Yaskawa INFORM job: R1_W27-A2(90,-90)POPR-KM-OK_MOD.JBI

/JOB
//NAME R1_W27-A2(90,-90)POPR-KM-OK_MOD
///FOLDERNAME KRIS-SCIANA
//POS
///NPOS 183,183,0,6,0,0
///TOOL 0
///POSTYPE PULSE
///PULSE
C00000=47255,92390,21974,-39561,97708,85383
C00001=10855,-90008,-88389,-33686,75537,85808
C00002=-111602,-139258,-125525,-5527,77988,-30584
C00003=-111602,-139258,-125525,-5527,77988,-30584
C00004=-63451,-99780,-87259,-34493,107645,-18593
C00005=-79235,-87779,-71168,-36428,98005,-22127
C00006=-81155,-88041,-68185,-36487,95587,-22123
C00007=-83679,-90006,-68978,-36755,94086,-22676
C00008=-83320,-89737,-68871,-36718,94298,-22597
C00009=-83320,-90271,-70181,-36754,94730,-22742
C00010=-84421,-91093,-70507,-36864,94080,-22984
C00011=-84421,-90731,-69628,-36842,93792,-22887
C00012=-81728,-89912,-71997,-36675,96467,-22659
C00013=-111602,-139258,-125525,-5527,77988,-30584
C00014=-111602,-139258,-125525,-5527,77988,-30584
C00015=-131748,-141016,-124490,10531,76516,-37016
C00016=-120565,-128207,-90021,8850,60749,-34228
C00017=-114295,-127384,-89205,7232,60054,-31882
C00018=-112834,-127008,-88848,6844,59902,-31333
C00019=-110412,-126666,-88756,6184,59829,-30410
C00020=-111525,-126835,-88802,6488,59856,-30835
C00021=-111525,-128465,-91197,6450,60489,-30798
C00022=-108910,-128023,-91079,5736,60447,-29805
C00023=-108910,-126871,-89375,5761,59994,-29827
C00024=-114109,-129808,-92766,7120,60979,-31753
C00025=-125724,-137992,-104372,9805,65099,-35816
C00026=-168598,-158328,-94882,65934,65859,5142
C00027=-138330,-90233,-84655,36621,76479,52498
C00028=-128715,-49536,-61129,33505,77884,56923
C00029=-128662,-48132,-55305,33830,75458,56202
C00030=-128776,-48721,-53911,34016,74532,55864
C00031=-127610,-48935,-54036,33707,74044,56192
C00032=-128384,-48797,-53955,33914,74367,55973
C00033=-127721,-49153,-57529,33460,75800,56690
C00034=-129344,-26255,-35376,41772,85568,55954
C00035=-129502,-28873,-35296,41846,84590,55492
C00036=-129628,-31082,-36795,41874,84489,55393
C00037=-129540,-29583,-35781,41856,84558,55460
C00038=-128070,-29028,-37630,41593,84938,56269
C00039=-125732,-38818,-42817,41353,82441,56314
C00040=-125732,-38715,-41972,41387,82085,56171
C00041=-125732,-38825,-42888,41351,82471,56325
C00042=-132576,-10372,-23557,42183,87769,55412
C00043=-126022,-12465,-28572,31920,86751,56828
C00044=-125240,-12576,-28656,31787,86457,57050
C00045=-126011,-12468,-28573,31917,86746,56832
C00046=-125354,-12526,-30294,30962,87436,57184
C00047=-120977,-16940,-33250,30218,85489,58339
C00048=-121063,-17240,-32162,30257,84802,58123
C00049=-121058,-15104,-30561,30253,84897,58149
C00050=-121061,-16554,-31651,30256,84834,58131
C00051=-121060,-15778,-32671,30227,85727,58368
C00052=-117907,-13652,-30768,29609,84558,59259
C00053=-117907,-13692,-29869,29630,84054,59130
C00054=-117057,-13593,-30324,29443,84053,59453
C00055=-124504,-18943,-37628,40859,87235,58732
C00056=-122503,-58034,-63350,23085,92729,-39111
C00057=-118561,-36204,-48728,23381,102965,-35613
C00058=-118381,-37612,-47396,23227,101492,-35840
C00059=-119514,-54944,-57534,22827,90064,-38535
C00060=-118197,-55011,-58807,22737,90395,-37994
C00061=-117359,-61105,-60828,21568,85220,-34341
C00062=-119392,-54872,-58672,22830,90711,-38368
C00063=-122456,-57021,-66004,23167,94704,-38710
C00064=-79548,-70371,-81102,-16241,84903,14397
C00065=-79548,-70265,-68951,-16505,77767,15353
C00066=-104563,-100291,-63220,13387,32000,-19094
C00067=-104975,-100452,-63184,13820,31966,-19359
C00068=-115302,-93136,-62932,26704,43721,-31733
C00069=-113448,-91077,-63180,22011,45608,-32160
C00070=-114452,-94731,-67163,22359,46409,-32454
C00071=-99886,-76150,-67523,500,65373,-23503
C00072=-75740,-68220,-64202,-17439,76767,16862
C00073=-76507,-66361,-64522,-17207,77706,16451
C00074=-95900,-77133,-67906,-2885,65671,-13753
C00075=-83981,-71880,-65491,-14621,70935,-768
C00076=-83123,-70857,-64909,-14849,71253,-493
C00077=-81635,-70718,-66741,-15162,72688,-135
C00078=-81323,-43477,-57369,-10673,89641,51992
C00079=-82758,-42773,-53931,-10445,87732,51670
C00080=-82626,-42173,-53561,-10465,87828,51707
C00081=-82621,-41471,-53126,-10465,87921,51700
C00082=-92310,-5151,-28231,-6661,90278,58032
C00083=-92716,-2727,-26257,-6592,90277,57898
C00084=-95848,18216,-9468,-2153,101928,56962
C00085=-96696,22336,-5572,-2620,102588,67876
C00086=-92622,2167,-26871,-6629,93158,57779
C00087=-102765,8643,-22555,7262,102808,72751
C00088=-102913,11884,-15167,7450,102139,72741
C00089=-104434,11036,-15928,7485,102306,72236
C00090=-104019,13462,-16416,6672,103835,72468
C00091=-100362,7840,-23814,352,99133,73837
C00092=-93505,-42567,-98732,-7157,86742,74535
C00093=-125724,-137992,-104372,9805,65099,-35816
C00094=-110950,-137574,-92834,6542,56798,-30799
C00095=-108633,-136098,-91409,5901,56506,-29909
C00096=-110317,-120133,-87198,6027,62209,-30244
C00097=-115536,-122151,-89589,7364,63072,-32157
C00098=-115536,-142518,-126484,6818,75223,-31432
C00099=-115536,-142518,-126484,6818,75223,-31432
C00100=27632,69086,-255,32308,94480,64498
C00101=22775,131727,30764,-8837,96794,84364
C00102=23208,121491,44257,-39062,86083,83812
C00103=-45129,13731,-11238,-25738,101470,44798
C00104=-54749,18539,-6974,-25294,98453,41899
C00105=-54749,18238,-2799,-25102,95977,42433
C00106=-54749,18226,-2184,-25080,95627,42508
C00107=-54749,18240,-2936,-25107,96054,42417
C00108=-50930,35725,13913,-25203,95936,43853
C00109=-64523,30372,3224,-1874,95567,42430
C00110=-64687,29964,2819,-1861,95602,42375
C00111=-65096,28955,1821,-1825,95689,42236
C00112=-64964,29394,1262,-1838,96260,42271
C00113=-65321,28613,-146,-1811,96720,42147
C00114=-68202,27629,-336,-1561,96271,41197
C00115=-68113,27223,145,-1567,95770,41232
C00116=-67724,25933,-1111,-1601,95888,41360
C00117=-68202,27629,-336,-1561,96271,41197
C00118=-69952,33819,5307,-1407,95949,40620
C00119=-71494,37291,10752,-1268,94359,40124
C00120=-71910,38959,12475,-1230,94150,39986
C00121=-71687,38230,9822,-1254,95411,40047
C00122=-69715,46382,18396,-1423,94355,40716
C00123=-70085,45287,18762,-1387,93560,40601
C00124=-70403,44519,17944,-1360,93663,40494
C00125=-69715,46382,18396,-1423,94355,40716
C00126=-70506,44470,16366,-1355,94608,40450
C00127=-74342,36127,7664,-1021,95621,39166
C00128=-67594,51845,26562,-12944,100620,40046
C00129=-67594,51857,27602,-12911,100003,40111
C00130=-67594,51846,26389,-12950,100725,40035
C00131=-74342,37093,2887,-1031,99056,39137
C00132=-67920,8103,-14728,-23481,111043,54078
C00133=-68371,9278,-10792,-23231,109243,54283
C00134=-71989,6025,-15002,-18365,107550,55075
C00135=-68543,9839,-10380,-23257,109228,54219
C00136=-67871,11157,-7953,-23050,108659,54597
C00137=-70618,6902,-11763,-25009,100838,46496
C00138=-68309,7669,-17399,-25439,105035,46441
C00139=-35319,67510,50034,-36864,102833,41158
C00140=-36426,60496,49514,-37352,95882,39315
C00141=-36245,61460,50947,-37306,95650,39472
C00142=-37635,75219,67177,-34434,97406,42519
C00143=-35605,73747,62011,-36095,100000,42690
C00144=-48748,75637,44138,-12559,109446,36491
C00145=-47018,7632,-18403,-16315,86685,22647
C00146=-48186,9094,-11222,-16117,82930,22742
C00147=-48900,12300,-7759,-15972,82326,22576
C00148=-48845,10311,-10218,-15969,82810,22529
C00149=-48144,8977,-10156,-16147,82248,22846
C00150=-48792,12294,-7764,-15997,82346,22611
C00151=-48554,12497,-7580,-16051,82384,22689
C00152=-47807,15110,-5208,-16221,82416,22944
C00153=-47830,15796,-4582,-16217,82378,22941
C00154=-47157,14640,-7349,-16336,83577,23014
C00155=-46490,6362,-16531,-16455,85053,23045
C00156=-51089,14800,-9249,10241,81305,-15900
C00157=-51639,15771,-6503,10417,80201,-16178
C00158=-51452,17933,-2732,10403,78988,-16218
C00159=-52394,14452,-5453,10658,78994,-16538
C00160=-51853,16186,-5099,10493,79587,-16303
C00161=-61783,45784,25403,13194,77537,-19938
C00162=-67433,89838,76993,23343,85040,-43070
C00163=-67406,90447,77765,23345,84883,-43090
C00164=-67651,91444,77676,23339,85475,-43066
C00165=-51787,16236,-7953,10429,81332,-16133
C00166=-102783,1332,-28831,-2508,120082,-77442
C00167=-102957,2789,-26573,-2528,119437,-77492
C00168=-103006,2286,-25832,-2518,118722,-77496
C00169=-103017,3676,-26663,-2555,119947,-77527
C00170=-103226,5472,-23865,-2576,119142,-77587
C00171=-101649,3064,-25171,-2232,118754,-76984
C00172=-101836,5087,-24653,-2291,119469,-77071
C00173=-102782,1324,-28838,-2508,120083,-77442
C00174=-102716,1959,-28722,-3690,98810,-77621
C00175=-111602,-139258,-125525,-5527,77988,-30584
C00176=-63451,-99780,-87259,-34493,107645,-18593
C00177=-77664,-93447,-72354,-35997,96893,-21092
C00178=-71109,-84007,-59579,-44165,102740,-19972
C00179=-76711,-72421,-54458,-45861,101920,-22309
C00180=-73740,-70290,-55538,-45661,104697,-22163
C00181=-73778,-73289,-89979,-52376,117942,-29543
C00182=4604,-97136,-110463,-3690,98810,-77621
BC00000=173361,170327,1069948
BC00001=285044,126360,1057855
BC00002=197925,2384,1013850
BC00003=398093,2384,1013850
BC00004=398093,2384,1013850
BC00005=398093,2384,1013850
BC00006=398093,2384,1013850
BC00007=398093,2384,1013850
BC00008=398093,2384,1013850
BC00009=398093,2384,1013850
BC00010=398093,2384,1013850
BC00011=398093,2384,1013850
BC00012=398093,2384,1013850
BC00013=398093,2384,1013850
BC00014=197925,2384,1013850
BC00015=16093,2384,1007970
BC00016=16093,2384,1007970
BC00017=16093,2384,1007970
BC00018=16093,2384,1007970
BC00019=16093,2384,1007970
BC00020=16093,2384,1007970
BC00021=16093,2384,1007970
BC00022=16093,2384,1007970
BC00023=16093,2384,1007970
BC00024=16093,2384,1007970
BC00025=16093,2384,1007970
BC00026=2663,3711,1022453
BC00027=269,7512,1047096
BC00028=269,7512,1047096
BC00029=269,7512,1047096
BC00030=269,7512,1047096
BC00031=269,7512,1047096
BC00032=269,7512,1047096
BC00033=269,7512,1047096
BC00034=15,11820,1075020
BC00035=15,11820,1075020
BC00036=15,11820,1075020
BC00037=15,11820,1075020
BC00038=15,11820,1075020
BC00039=15,11820,1075020
BC00040=15,11820,1075020
BC00041=15,11820,1075020
BC00042=15,11820,1075020
BC00043=15,11820,1075020
BC00044=15,11820,1075020
BC00045=15,11820,1075020
BC00046=15,11820,1075020
BC00047=15,11820,1075020
BC00048=15,11820,1075020
BC00049=15,11820,1075020
BC00050=15,11820,1075020
BC00051=15,11820,1075020
BC00052=15,11820,1075020
BC00053=15,11820,1075020
BC00054=15,11820,1075020
BC00055=15,11820,1075020
BC00056=15,49099,1075175
BC00057=15,47349,1075175
BC00058=15,47349,1075175
BC00059=15,47349,1075175
BC00060=15,47349,1075175
BC00061=15,62077,1075175
BC00062=15,62577,1075175
BC00063=15,63827,1075175
BC00064=15,12213,1075175
BC00065=15,12213,1075175
BC00066=16,12213,1075171
BC00067=16,12213,1075171
BC00068=16,12213,1075171
BC00069=16,12213,1075171
BC00070=16,12213,1075171
BC00071=16,12213,1075171
BC00072=15,16755,1075175
BC00073=15,16755,1075175
BC00074=16,12213,1075171
BC00075=16,12213,1075171
BC00076=16,12213,1075171
BC00077=16,12213,1075171
BC00078=16,12213,1075171
BC00079=16,12213,1075171
BC00080=16,12213,1075171
BC00081=16,12213,1075171
BC00082=16,12213,1075171
BC00083=16,12213,1075171
BC00084=16,12213,1075171
BC00085=16,12213,1075171
BC00086=16,12213,1075171
BC00087=17,22433,1075169
BC00088=17,22433,1075167
BC00089=17,22433,1075167
BC00090=17,22433,1075169
BC00091=16,12213,1075171
BC00092=16,12213,1075171
BC00093=16093,2384,1007970
BC00094=16093,2384,1007970
BC00095=16093,2384,1007970
BC00096=16093,2384,1007970
BC00097=16093,2384,1007970
BC00098=16093,2384,1007970
BC00099=92875,102,1007970
BC00100=25030,15919,1060143
BC00101=103306,16446,1075157
BC00102=79646,13110,1075161
BC00103=246913,5043,1075175
BC00104=246913,5043,1075175
BC00105=246913,5043,1075175
BC00106=246913,5043,1075175
BC00107=246913,5043,1075175
BC00108=246913,5043,1075175
BC00109=246913,5043,1075175
BC00110=246913,5043,1075175
BC00111=246913,5043,1075175
BC00112=246913,5043,1075175
BC00113=246913,5043,1075175
BC00114=246913,5043,1075175
BC00115=246913,5043,1075175
BC00116=246913,5043,1075175
BC00117=246913,5043,1075175
BC00118=246913,5043,1075175
BC00119=246913,5043,1075175
BC00120=246913,5043,1075175
BC00121=246913,5043,1075175
BC00122=246913,5043,1075175
BC00123=246913,5043,1075175
BC00124=246913,5043,1075175
BC00125=246913,5043,1075175
BC00126=246913,5043,1075175
BC00127=246913,5043,1075175
BC00128=246913,5043,1075175
BC00129=246913,5043,1075175
BC00130=246913,5043,1075175
BC00131=246913,5043,1075175
BC00132=310215,25331,1075175
BC00133=304559,24148,1075175
BC00134=304559,24148,1075175
BC00135=302296,23674,1075175
BC00136=302296,23674,1075175
BC00137=304559,24148,1075175
BC00138=304559,24148,1075175
BC00139=197323,15,1075175
BC00140=197323,15,1075175
BC00141=197323,15,1075175
BC00142=197323,15,1075175
BC00143=197323,15,1075175
BC00144=197323,15,1075175
BC00145=197986,15,1075175
BC00146=197986,15,1075175
BC00147=198112,15,1075175
BC00148=198252,15,1075175
BC00149=198252,15,1075175
BC00150=198112,15,1075175
BC00151=198112,15,1075175
BC00152=198112,15,1075175
BC00153=198112,15,1075175
BC00154=198112,15,1075175
BC00155=199434,15,1075175
BC00156=148787,33401,1075175
BC00157=154351,32151,1075175
BC00158=155733,31841,1075173
BC00159=156576,31651,1075175
BC00160=156576,31651,1075175
BC00161=155733,31841,1075173
BC00162=155733,31841,1075173
BC00163=155733,31841,1075173
BC00164=155733,31841,1075173
BC00165=148927,71500,1075175
BC00166=344706,64580,1052547
BC00167=343940,58320,1037184
BC00168=343871,57754,1035794
BC00169=343634,55816,1031039
BC00170=343634,55816,1031039
BC00171=343871,57754,1035794
BC00172=343871,57754,1035794
BC00173=341638,64598,1052619
BC00174=341637,64597,1052617
BC00175=398093,160168,1013850
BC00176=398093,2384,1013850
BC00177=398093,2384,1013850
BC00178=398093,2384,1013850
BC00179=398093,2384,1013850
BC00180=398093,2384,1013850
BC00181=398093,2384,1013850
BC00182=176985,505314,1052617
///POSTYPE BASE
///RECTAN
///RCONF 0,0,0,0,1,0,0,0,0,0,0,0,0,0,0,0,0,0,0,0,0,0,0,0
P00006=2.006,1.622,-0.565,0.0000,0.0000,0.0000
///RCONF 0,0,0,0,0,0,0,0,0,0,0,0,0,0,0,0,0,0,0,0,0,0,0,0
P00023=-2.957,-4.083,2.762,0.0000,0.0000,0.0000
P00024=-1.466,-0.226,-0.419,0.0000,0.0000,0.0000
P00025=3.643,0.007,-2.585,0.0000,0.0000,0.0000
P00040=2.716,-0.016,3.014,0.0000,0.0000,0.0000
P00041=-0.109,0.014,0.966,0.0000,0.0000,0.0000
//INST
///DATE 2025/01/17 12:20
///ATTR SC,RW
///GROUP1 RB1,BS1
NOP
SFTOF
MOVJ C00000 BC00000 VJ=100.00
MOVJ C00001 BC00001 VJ=100.00
MOVJ C00002 BC00002 VJ=100.00
'DODANO BP 060624
MOVJ C00003 BC00003 VJ=100.00
MOVJ C00004 BC00004 VJ=100.00
MOVL C00005 BC00005 V=233.3
MOVL C00006 BC00006 V=60.0
REFP 3 C00007 BC00007
CALL JOB:SEARCH-R1
SET P040 P006
SFTON P040
MOVL C00008 BC00008 V=100.0
MOVL C00009 BC00009 V=100.0
MOVL C00010 BC00010 V=60.0
REFP 3 C00011 BC00011
CALL JOB:SEARCH-R1
SET P040 P006
SFTON P040
MOVL C00012 BC00012 V=100.0
MOVJ C00013 BC00013 VJ=100.00
MOVJ C00014 BC00014 VJ=100.00
MOVL C00015 BC00015 V=666.7
MOVL C00016 BC00016 V=666.7
MOVL C00017 BC00017 V=233.3
MOVL C00018 BC00018 V=60.0
REFP 3 C00019 BC00019
CALL JOB:SEARCH-R1
SET P041 P006
SFTON P041
MOVL C00020 BC00020 V=100.0
MOVL C00021 BC00021 V=100.0
MOVL C00022 BC00022 V=60.0
REFP 3 C00023 BC00023
CALL JOB:SEARCH-R1
SET P041 P006
SFTON P041
MOVL C00024 BC00024 V=100.0
MOVL C00025 BC00025 V=666.7
'KONIEC BP 060624
MOVJ C00026 BC00026 VJ=100.00
MOVJ C00027 BC00027 VJ=100.00
MOVJ C00028 BC00028 VJ=100.00
MOVJ C00029 BC00029 VJ=100.00
MOVL C00030 BC00030 V=60.0
REFP 3 C00031 BC00031
CALL JOB:SEARCH-R1
SET P023 P006
SFTON P023
MOVL C00032 BC00032 V=60.0
MOVL C00033 BC00033 V=100.0
MOVL C00034 BC00034 V=100.0
MOVL C00035 BC00035 V=100.0
REFP 3 C00036 BC00036
CALL JOB:SEARCH-R1
SET P023 P006
SFTON P023
MOVL C00037 BC00037 V=60.0
MOVL C00038 BC00038 V=100.0
MOVL C00039 BC00039 V=100.0
REFP 3 C00040 BC00040
CALL JOB:SEARCH-R1
SET P023 P006
SFTON P023
MOVL C00041 BC00041 V=60.0
'DRUGI NOWY POMIAR
SFTOF
MOVL C00042 BC00042 V=100.0
MOVL C00043 BC00043 V=100.0
REFP 3 C00044 BC00044
CALL JOB:SEARCH-R1
SET P024 P006
SFTON P024
MOVL C00045 BC00045 V=60.0
MOVL C00046 BC00046 V=100.0
MOVL C00047 BC00047 V=100.0
MOVL C00048 BC00048 V=60.0
REFP 3 C00049 BC00049
CALL JOB:SEARCH-R1
SET P024 P006
SFTON P024
MOVL C00050 BC00050 V=60.0
MOVL C00051 BC00051 V=100.0
MOVL C00052 BC00052 V=60.0
REFP 3 C00053 BC00053
CALL JOB:SEARCH-R1
SET P024 P006
SFTON P024
MOVL C00054 BC00054 V=60.0
MOVJ C00055 BC00055 VJ=30.00
SFTOF
COMM 'Path W988
COMM SFTOF
COMM SFTON P023
COMM CALL JOB:COFNIJ_DRUT
COMM MOVJ C00056 BC00056 VJ=50.00
COMM MOVJ C00057 BC00057 VJ=100.00
COMM MOVL C00058 BC00058 V=100.0 PL=0
COMM REFP 1 C00059 BC00059
COMM REFP 2 C00060 BC00060
COMM MACRO1 MJ#(0) ARGF7
COMM ARCON
COMM SFTON P024
COMM MOVL C00061 BC00061 V=10.8
COMM ARCOF
COMM MOVL C00062 BC00062 V=100.0
COMM MOVJ C00063 BC00063 VJ=50.00
COMM SFTOF
COMM 'Path W989
COMM SFTOF
SFTON P023
MOVJ C00064 BC00064 VJ=100.00
MOVJ C00065 BC00065 VJ=50.00
MOVL C00066 BC00066 V=100.0
ARCON
MOVL C00067 BC00067 V=8.3
MOVL C00068 BC00068 V=8.3
MOVL C00069 BC00069 V=8.3
ARCOF
SFTOF
MOVL C00070 BC00070 V=83.3
SFTON P023
MOVL C00071 BC00071 V=100.0 PL=0
REFP 1 C00072 BC00072
REFP 2 C00073 BC00073
MACRO1 MJ#(0) ARGF7
ARCON
TIMER T=0.50
MOVL C00074 BC00074 V=10.0
MOVL C00075 BC00075 V=10.0
MOVL C00076 BC00076 V=10.0
ARCOF
MOVJ C00077 BC00077 VJ=15.00
MOVJ C00078 BC00078 VJ=100.00
MOVJ C00079 BC00079 VJ=20.00 PL=0
ARCON
MOVL C00080 BC00080 V=10.0
MOVL C00081 BC00081 V=10.0
SFTON P024
MOVL C00082 BC00082 V=10.0
MOVL C00083 BC00083 V=10.0
MOVL C00084 BC00084 V=13.3
MOVL C00085 BC00085 V=13.3
ARCOF
MOVJ C00086 BC00086 VJ=15.00
MOVJ C00087 BC00087 VJ=100.00
MOVJ C00088 BC00088 VJ=20.00 PL=0
ARCON
MOVL C00089 BC00089 V=10.0
ARCOF
MOVL C00090 BC00090 V=100.0
MOVL C00091 BC00091 V=166.7
MOVJ C00092 BC00092 VJ=100.00
SFTOF
'BP 060624
MOVJ C00093 BC00093 VJ=100.00
MOVJ C00094 BC00094 VJ=100.00
SFTON P041
MOVL C00095 BC00095 V=100.0 PL=0
MACRO1 MJ#(0) ARGF6
ARCON
MOVL C00096 BC00096 V=11.7
ARCOF
MOVL C00097 BC00097 V=11.7
SFTOF
MOVL C00098 BC00098 V=666.7
MOVL C00099 BC00099 V=666.7
'KONIEC BP 060624
'2 STRONA
MOVJ C00100 BC00100 VJ=100.00
'Path VIA1124
SFTOF
MOVJ C00101 BC00101 VJ=100.00
CALL JOB:ONLYCUT-R1_LONG
'Path S992
SFTOF
MOVJ C00102 BC00102 VJ=100.00
SFTOF
MOVJ C00103 BC00103 VJ=100.00
MOVJ C00104 BC00104 VJ=100.00
MOVL C00105 BC00105 V=83.3
REFP 3 C00106 BC00106
CALL JOB:SEARCH-R1
SET P024 P006
SFTON P024
MOVL C00107 BC00107 V=166.7
MOVL C00108 BC00108 V=166.7
MOVL C00109 BC00109 V=166.7
MOVL C00110 BC00110 V=166.7
REFP 3 C00111 BC00111
CALL JOB:SEARCH-R1
SET P024 P006
SFTON P024
MOVL C00112 BC00112 V=166.7
MOVL C00113 BC00113 V=166.7
MOVL C00114 BC00114 V=166.7
MOVL C00115 BC00115 V=166.7
REFP 3 C00116 BC00116
CALL JOB:SEARCH-R1
SET P024 P006
SFTON P024
MOVL C00117 BC00117 V=166.7
SFTOF
MOVL C00118 BC00118 V=166.7
MOVL C00119 BC00119 V=166.7
REFP 3 C00120 BC00120
CALL JOB:SEARCH-R1
SET P025 P006
SFTON P025
MOVL C00121 BC00121 V=166.7
MOVL C00122 BC00122 V=166.7
MOVL C00123 BC00123 V=166.7
REFP 3 C00124 BC00124
CALL JOB:SEARCH-R1
SET P025 P006
SFTON P025
MOVL C00125 BC00125 V=166.7
MOVL C00126 BC00126 V=166.7
MOVL C00127 BC00127 V=166.7
MOVL C00128 BC00128 V=166.7
REFP 3 C00129 BC00129
CALL JOB:SEARCH-R1
SET P025 P006
SFTON P025
MOVL C00130 BC00130 V=166.7
MOVL C00131 BC00131 V=166.7
COMM 'Path W993
COMM SFTOF
COMM SFTON P024
COMM MOVJ C00132 BC00132 VJ=100.00
COMM MOVJ C00133 BC00133 VJ=100.00
COMM SFTON P024
COMM MOVL C00134 BC00134 V=100.0 PL=0
COMM REFP 1 C00135 BC00135
COMM REFP 2 C00136 BC00136
COMM MACRO1 MJ#(0) ARGF7
COMM ARCON
COMM SFTON P025
COMM MOVL C00137 BC00137 V=10.0
COMM ARCOF
COMM MOVL C00138 BC00138 V=100.0
COMM SFTOF
SFTON P024
MOVJ C00139 BC00139 VJ=20.00
MOVJ C00140 BC00140 VJ=20.00 PL=0
ARCON
MOVL C00141 BC00141 V=8.3
MOVL C00142 BC00142 V=8.3
ARCOF
MOVL C00143 BC00143 V=83.3
MOVJ C00144 BC00144 VJ=20.00
MOVJ C00145 BC00145 VJ=20.00
MOVJ C00146 BC00146 VJ=100.00
SFTON P024
MOVL C00147 BC00147 V=100.0 PL=0
REFP 1 C00148 BC00148
REFP 2 C00149 BC00149
MACRO1 MJ#(0) ARGF7
ARCON
MOVL C00150 BC00150 V=10.0
MOVL C00151 BC00151 V=10.0
MOVL C00152 BC00152 V=10.0
MOVL C00153 BC00153 V=10.0
ARCOF
MOVL C00154 BC00154 V=166.7
MOVL C00155 BC00155 V=166.7
SFTOF
'Path W995
SFTOF
SFTON P024
MOVJ C00156 BC00156 VJ=100.00
MOVJ C00157 BC00157 VJ=100.00
SFTON P024
MOVL C00158 BC00158 V=100.0 PL=0
REFP 1 C00159 BC00159
REFP 2 C00160 BC00160
MACRO1 MJ#(0) ARGF7
ARCON
SFTON P025
MOVL C00161 BC00161 V=10.0
MOVL C00162 BC00162 V=13.3
MOVL C00163 BC00163 V=13.3
ARCOF
MOVL C00164 BC00164 V=400.0
MOVL C00165 BC00165 V=1000.0
SFTOF
MOVJ C00166 BC00166 VJ=100.00
MOVJ C00167 BC00167 VJ=100.00
SFTON P025
MOVL C00168 BC00168 V=100.0 PL=0
REFP 1 C00169 BC00169
REFP 2 C00170 BC00170
MACRO1 MJ#(0) ARGF7
ARCON
MOVL C00171 BC00171 V=10.0
ARCOF
MOVL C00172 BC00172 V=166.7
MOVL C00173 BC00173 V=400.0
SFTOF
MOVJ C00174 BC00174 VJ=100.00
'BP 060624
SFTOF
MOVL C00175 BC00175 V=666.7
MOVL C00176 BC00176 V=666.7
MOVL C00177 BC00177 V=666.7
SFTON P040
MOVL C00178 BC00178 V=100.0 PL=0
MACRO1 MJ#(0) ARGF6
ARCON
MOVL C00179 BC00179 V=11.7
ARCOF
MOVL C00180 BC00180 V=266.7
SFTOF
MOVJ C00181 BC00181 VJ=100.00
'KONIEC BP 060624
MOVJ C00182 BC00182 VJ=100.00
END
